PROGRAM o_Cons_Cmd_Actionneurs
VAR
	Calcul_Temp1: REAL;
	Mode_NEP_Chaud: BOOL;
	Mode_NEP_Froid: BOOL;
	Calcul_Debit_Bypass: REAL;
	ACH_Deb_Souf_Etat_Depol: REAL;
	ACH_Deb_Souf_Etat_Libre: REAL;
	ACH_Mode_Auto_Out_Debit_Souf: REAL;
	Consigne_Mode_EnFctnmnt_PD: REAL := 67.0;
	Consigne_Mode_EnFctnmnt_GD: REAL := 600.0;
END_VAR

(**********************************************Commande des actionneurs*)
Cmd_Appli_PC_Cab					:= (Mode_Auto.Cmd_Prise  AND Mode_Auto.Enable) OR (Mode_Manu.Cmd_Prise AND Mode_Manu.Enable);
Cmd_Appli_Vanne_Alim_Douche			:= (Mode_Auto.Cmd_Douche  AND Mode_Auto.Enable) OR (Mode_Manu.Cmd_Douche AND Mode_Manu.Enable) OR Forc_Ouv_Alim_Lav_Dou;
Cmd_Appli_Vanne_Alim_Douchette		:= ((Mode_Auto.Cmd_Douchette  AND Mode_Auto.Enable) OR (Mode_Manu.Cmd_Douchette AND Mode_Manu.Enable) OR Mode_Cabine_Nettoyage);
Cmd_Appli_Vanne_Alim_Lavabo			:= (Mode_Auto.Cmd_Lavabo  AND Mode_Auto.Enable) OR (Mode_Manu.Cmd_Lavabo AND Mode_Manu.Enable);
Cmd_Appli_Vanne_Vid_Douche			:= ((Mode_Auto.Cmd_Vidange_Douche  AND Mode_Auto.Enable) OR (Mode_Manu.Cmd_Vidange_Douche AND Mode_Manu.Enable) OR Mode_Cabine_Nettoyage);
Cmd_Appli_Vanne_Vid_Lavabo			:= ((Mode_Auto.Cmd_Vidange_Lavabo  AND Mode_Auto.Enable) OR (Mode_Manu.Cmd_Vidange_Lavabo AND Mode_Manu.Enable) OR Mode_Cabine_Nettoyage);
Cmd_Appli_ElectroValve_Alim_Douche	:= (Mode_Auto.Cmd_Electrovanne_Douche  AND Mode_Auto.Enable) OR (Mode_Manu.Cmd_Electrovanne_Douche AND Mode_Manu.Enable);
Cmd_Appli_ElectroValve_Alim_Lavabo	:= (Mode_Auto.Cmd_Electrovanne_Lavabo  AND Mode_Auto.Enable) OR (Mode_Manu.Cmd_Electrovanne_Lavabo AND Mode_Manu.Enable) OR Forc_Ouv_Alim_Lav_Dou;
Cmd_Appli_Reg_Etanche_Souf			:= (Cons_Actionneur_Registre_Souf_m3h > ((Cons_Max_Bas_Deb_Ext + 0.5) * Volume_Cabine)) AND Option_Reg_Etanche_Souf;
Cmd_Appli_Vanne_Alim_NEP			:=  (Mode_Auto.Cmd_NEP  AND Mode_Auto.Enable) OR (Mode_Manu.Cmd_NEP AND Mode_Manu.Enable);
Cmd_Appli_Verin_WC_GV				:=(Mode_Auto.Cmd_Verin_WC_GV  AND Mode_Auto.Enable) OR (Mode_Manu.Cmd_Verin_WC_GV AND Mode_Manu.Enable);
Cmd_Appli_Verin_WC_PV				:=(Mode_Auto.Cmd_Verin_WC_PV  AND Mode_Auto.Enable) OR (Mode_Manu.Cmd_Verin_WC_PV AND Mode_Manu.Enable);

(*Convertion des valeurs m3/h en Vol/h (ACH)*)
ACH_Deb_Souf_Etat_Depol 	:= Cons_Deb_Souf_Etat_Depol * Volume_Cabine;
ACH_Deb_Souf_Etat_Libre 	:= Cons_Deb_Souf_Etat_Libre * Volume_Cabine;
ACH_Mode_Auto_Out_Debit_Souf:= Mode_Auto.Out_Debit_Souf * Volume_Cabine;

(**********************************************Gestion de la consigne de débit en état cabine libre*)
IF(Mode_Cabine_Libre)
	THEN
	Cons_Actionneur_Registre_Ext_Volh 					:= ACH_Deb_Souf_Etat_Libre;
	Cons_Actionneur_Registre_Souf_Volh 					:= ACH_Deb_Souf_Etat_Libre;
	
	IF (ACH_Deb_Souf_Etat_Libre < 354.0) //Mettre la valeur maximum du débit du registre en diam 100mm
		THEN
		GVL_RegTROX.ConsAppliDeb_RegSouf_GD_FCVT01		:= 0.0;
		GVL_RegTROX.ConsAppliDeb_RegSouf_PD_FCVT02		:= ACH_Deb_Souf_Etat_Libre;
		ELSE
		GVL_RegTROX.ConsAppliDeb_RegSouf_GD_FCVT01		:= ACH_Deb_Souf_Etat_Libre;
		GVL_RegTROX.ConsAppliDeb_RegSouf_PD_FCVT02		:= 0.0;	
	END_IF
	GVL_RegTROX.ConsAppliDeb_RegSouf_Cabine_FCVT03		:= 1020.0; //Mettre le débit maximum pour qu'il reste ouvert à 100%
	GVL_RegTROX.ConsAppliDeb_Reg_Bypass_FCVT04			:= 0.0;
	GVL_RegTROX.ConsAppliDeb_RegSouf_CabGD_FCVT05		:= 0.0;
	GVL_RegTROX.ConsAppliDeb_RegSouf_CabPD_FCVT06		:= 0.0;
	GVL_RegTROX.ConsAppliDeb_RegRep_FCVT07				:= 0.0;
END_IF;

(**********************************************Gestion de la consigne de débit en etat cabine dépollution*)
IF(Mode_Cabine_Depollution OR Mode_Depollution_cycle1)
	THEN
	IF (Mode_Depollution_cycle1) // 1er cycle, décontamination de la CTA
		THEN
		Cons_Actionneur_Registre_Ext_Volh 					:= ACH_Deb_Souf_Etat_Depol;
		Cons_Actionneur_Registre_Souf_Volh 					:= ACH_Deb_Souf_Etat_Depol;
		
		GVL_RegTROX.ConsAppliDeb_RegSouf_GD_FCVT01			:= 375.0;
		GVL_RegTROX.ConsAppliDeb_RegSouf_PD_FCVT02			:= 100.0;
		GVL_RegTROX.ConsAppliDeb_RegSouf_Cabine_FCVT03		:= 0.0;
		GVL_RegTROX.ConsAppliDeb_Reg_Bypass_FCVT04			:= 0.0;
		GVL_RegTROX.ConsAppliDeb_RegSouf_CabGD_FCVT05		:= 575.0;
		GVL_RegTROX.ConsAppliDeb_RegSouf_CabPD_FCVT06		:= 100.0;
		GVL_RegTROX.ConsAppliDeb_RegRep_FCVT07				:= 200.0;
	END_IF;
	IF (Mode_Cabine_Depollution AND NOT Mode_Depollution_cycle1) // 2ème cycle, décontamination de la cabine
		THEN
		Cons_Actionneur_Registre_Ext_Volh 					:= ACH_Deb_Souf_Etat_Depol;
		Cons_Actionneur_Registre_Souf_Volh 					:= ACH_Deb_Souf_Etat_Depol;
		
		GVL_RegTROX.ConsAppliDeb_RegSouf_GD_FCVT01			:= ACH_Deb_Souf_Etat_Depol;
		GVL_RegTROX.ConsAppliDeb_RegSouf_PD_FCVT02			:= 0.0;
		GVL_RegTROX.ConsAppliDeb_RegSouf_Cabine_FCVT03		:= 1020.0; //Mettre le débit maximum pour qu'il reste ouvert à 100%
		GVL_RegTROX.ConsAppliDeb_Reg_Bypass_FCVT04			:= 0.0;
		GVL_RegTROX.ConsAppliDeb_RegSouf_CabGD_FCVT05		:= 0.0;
		GVL_RegTROX.ConsAppliDeb_RegSouf_CabPD_FCVT06		:= 0.0;
		GVL_RegTROX.ConsAppliDeb_RegRep_FCVT07				:= 0.0;
	END_IF;
END_IF;

(**********************************************Gestion de la consigne de débit en etat cabine Mode mise en condition*)
IF(Mode_MEnCond AND NOT Mode_Cabine_Libre)
	THEN
	Cons_Actionneur_Registre_Ext_Volh 					:= ACH_Mode_Auto_Out_Debit_Souf;
	Cons_Actionneur_Registre_Souf_Volh 					:= ACH_Mode_Auto_Out_Debit_Souf;
	
	GVL_RegTROX.ConsAppliDeb_RegSouf_GD_FCVT01			:= 0.0;
	GVL_RegTROX.ConsAppliDeb_RegSouf_PD_FCVT02			:= 0.0;
	GVL_RegTROX.ConsAppliDeb_RegSouf_Cabine_FCVT03		:= 0.0;
	GVL_RegTROX.ConsAppliDeb_Reg_Bypass_FCVT04			:= 0.0;
	IF (ACH_Mode_Auto_Out_Debit_Souf < 354.0)  //Mettre la valeur maximum du débit du registre en diam 100mm
		THEN
		GVL_RegTROX.ConsAppliDeb_RegSouf_CabGD_FCVT05	:= 0.0;
		GVL_RegTROX.ConsAppliDeb_RegSouf_CabPD_FCVT06	:= ACH_Mode_Auto_Out_Debit_Souf;
		ELSE
		GVL_RegTROX.ConsAppliDeb_RegSouf_CabGD_FCVT05	:= ACH_Mode_Auto_Out_Debit_Souf;
		GVL_RegTROX.ConsAppliDeb_RegSouf_CabPD_FCVT06	:= 0.0;	
	END_IF
	GVL_RegTROX.ConsAppliDeb_RegRep_FCVT07				:= 1020.0; //Mettre le débit maximum pour qu'il reste ouvert à 100%
END_IF;

(**********************************************Gestion de la consigne de débit en etat cabine Mode fonctionnement*)
IF(Mode_Fctnmt AND NOT Mode_Cabine_Libre)
	THEN
	Cons_Actionneur_Registre_Ext_Volh 					:= ACH_Mode_Auto_Out_Debit_Souf;
	Cons_Actionneur_Registre_Souf_Volh 					:= ACH_Mode_Auto_Out_Debit_Souf;
	(*IF (ACH_Mode_Auto_Out_Debit_Souf < 354.0) //Mettre la valeur maximum du débit du registre en diam 100mm
		THEN
		GVL_RegTROX.ConsAppliDeb_RegSouf_GD_FCVT01		:= 0.0;
		GVL_RegTROX.ConsAppliDeb_RegSouf_PD_FCVT02		:= ACH_Mode_Auto_Out_Debit_Souf;
		ELSE
		GVL_RegTROX.ConsAppliDeb_RegSouf_GD_FCVT01		:= ACH_Mode_Auto_Out_Debit_Souf;
		GVL_RegTROX.ConsAppliDeb_RegSouf_PD_FCVT02		:= 0.0;	
	END_IF*)
	GVL_RegTROX.ConsAppliDeb_RegSouf_GD_FCVT01			:= 0.0;
	GVL_RegTROX.ConsAppliDeb_RegSouf_PD_FCVT02			:= ACH_Mode_Auto_Out_Debit_Souf;
	GVL_RegTROX.ConsAppliDeb_RegSouf_Cabine_FCVT03		:= 0.0;
	Calcul_Debit_Bypass 								:= LIMIT(0.0, 600.0 - (Consigne_Mode_EnFctnmnt_GD + ACH_Mode_Auto_Out_Debit_Souf), 579.0);
	GVL_RegTROX.ConsAppliDeb_Reg_Bypass_FCVT04			:= Calcul_Debit_Bypass;
	GVL_RegTROX.ConsAppliDeb_RegSouf_CabGD_FCVT05		:= Consigne_Mode_EnFctnmnt_GD;
	GVL_RegTROX.ConsAppliDeb_RegSouf_CabPD_FCVT06		:= 0.0;
	(*IF (ACH_Mode_Auto_Out_Debit_Souf < 354.0) //Mettre la valeur maximum du débit du registre en diam 100mm
		THEN
		GVL_RegTROX.ConsAppliDeb_RegSouf_CabGD_FCVT05	:= 0.0;
		GVL_RegTROX.ConsAppliDeb_RegSouf_CabPD_FCVT06	:= ACH_Mode_Auto_Out_Debit_Souf;
		ELSE
		GVL_RegTROX.ConsAppliDeb_RegSouf_CabGD_FCVT05	:= ACH_Mode_Auto_Out_Debit_Souf;
		GVL_RegTROX.ConsAppliDeb_RegSouf_CabPD_FCVT06	:= 0.0;	
	END_IF*)
	GVL_RegTROX.ConsAppliDeb_RegRep_FCVT07				:= LIMIT(0, Consigne_Mode_EnFctnmnt_GD - ACH_Mode_Auto_Out_Debit_Souf, 1020.0);
END_IF;

(**********************************************Consigne des actionneurs en mode manuel*)
IF(Mode_Cabine_Manuel)
	THEN
	Cons_Actionneur_Registre_Ext_Volh 					:= Cons_Deb_Soufflage_Appli;
	Cons_Actionneur_Registre_Souf_Volh 					:= Cons_Deb_Soufflage_Appli;
	IF (Cons_Deb_Soufflage_Appli < 354.0) //Mettre la valeur maximum du débit du registre en diam 100mm
		THEN
		GVL_RegTROX.ConsAppliDeb_RegSouf_GD_FCVT01		:= 0.0;
		GVL_RegTROX.ConsAppliDeb_RegSouf_PD_FCVT02		:= Cons_Deb_Soufflage_Appli;
		ELSE
		GVL_RegTROX.ConsAppliDeb_RegSouf_GD_FCVT01		:= Cons_Deb_Soufflage_Appli;
		GVL_RegTROX.ConsAppliDeb_RegSouf_PD_FCVT02		:= 0.0;	
	END_IF
	GVL_RegTROX.ConsAppliDeb_RegSouf_Cabine_FCVT03		:= 0.0;
	GVL_RegTROX.ConsAppliDeb_Reg_Bypass_FCVT04			:= 0.0;
	GVL_RegTROX.ConsAppliDeb_RegSouf_CabGD_FCVT05		:= 0.0;
	GVL_RegTROX.ConsAppliDeb_RegSouf_CabPD_FCVT06		:= 0.0;
	GVL_RegTROX.ConsAppliDeb_RegRep_FCVT07				:= 0.0;
END_IF;

(**********************************************Gestion des consignes en cas de défaut sur le capteur de pression*)
IF (Defaut_Sonde_Press_Cabine AND NOT Dmd_Post_Ventilation)
	THEN
	GVL_RegTROX.ConsAppliDeb_RegSouf_GD_FCVT01			:= 0.0;
	GVL_RegTROX.ConsAppliDeb_RegSouf_PD_FCVT02			:= 0.0;	
	GVL_RegTROX.ConsAppliDeb_RegSouf_Cabine_FCVT03		:= 0.0;
	GVL_RegTROX.ConsAppliDeb_Reg_Bypass_FCVT04			:= 0.0;
	GVL_RegTROX.ConsAppliDeb_RegSouf_CabGD_FCVT05		:= 0.0;
	GVL_RegTROX.ConsAppliDeb_RegSouf_CabPD_FCVT06		:= 0.0;
	GVL_RegTROX.ConsAppliDeb_RegRep_FCVT07				:= 0.0;
END_IF

(**********************************************Consigne des actionneurs en mode automatique*)
IF(Mode_Cabine_Automatique AND NOT Mode_Cabine_Depollution AND NOT Mode_MEnCond AND NOT Mode_Fctnmt)
	THEN
	Cons_Actionneur_Registre_Ext_Volh	:= Cons_Deb_Soufflage_Appli;
	Cons_Actionneur_Registre_Souf_Volh	:= Cons_Deb_Soufflage_Appli;
	Cons_Actionneur_Moteur_ByPass		:= Mode_Auto.Out_Cons_Moteur_ByPass;
	// Deux types de fonctionnement, la première si une reccette est déclaré avec une gestion de CTA et le deuxième type sans gestion de CTA
	IF (RS_MEnCond.Q1)// gestion avec CTA (Activation des redistres de soufflage générale et du soufflage de la cabine)
		THEN
		Cons_Actionneur_Registre_Ext_Volh 					:= ACH_Mode_Auto_Out_Debit_Souf;
		Cons_Actionneur_Registre_Souf_Volh 					:= ACH_Mode_Auto_Out_Debit_Souf;
		(*IF (ACH_Mode_Auto_Out_Debit_Souf < 354.0) //Mettre la valeur maximum du débit du registre en diam 100mm
			THEN
			GVL_RegTROX.ConsAppliDeb_RegSouf_GD_FCVT01		:= 0.0;
			GVL_RegTROX.ConsAppliDeb_RegSouf_PD_FCVT02		:= ACH_Mode_Auto_Out_Debit_Souf;
			ELSE
			GVL_RegTROX.ConsAppliDeb_RegSouf_GD_FCVT01		:= ACH_Mode_Auto_Out_Debit_Souf;
			GVL_RegTROX.ConsAppliDeb_RegSouf_PD_FCVT02		:= 0.0;	
		END_IF*)
		GVL_RegTROX.ConsAppliDeb_RegSouf_GD_FCVT01			:= 0.0;
		GVL_RegTROX.ConsAppliDeb_RegSouf_PD_FCVT02			:= Consigne_Mode_EnFctnmnt_PD;
		GVL_RegTROX.ConsAppliDeb_RegSouf_Cabine_FCVT03		:= 0.0;
		Calcul_Debit_Bypass 								:= LIMIT(0.0, 600.0 - (Consigne_Mode_EnFctnmnt_GD + Consigne_Mode_EnFctnmnt_PD), 579.0);
		GVL_RegTROX.ConsAppliDeb_Reg_Bypass_FCVT04			:= Calcul_Debit_Bypass;
		GVL_RegTROX.ConsAppliDeb_RegSouf_CabGD_FCVT05		:= Consigne_Mode_EnFctnmnt_GD;
		GVL_RegTROX.ConsAppliDeb_RegSouf_CabPD_FCVT06		:= 0.0;
		(*IF (ACH_Mode_Auto_Out_Debit_Souf < 354.0) //Mettre la valeur maximum du débit du registre en diam 100mm
			THEN
			GVL_RegTROX.ConsAppliDeb_RegSouf_CabGD_FCVT05	:= 0.0;
			GVL_RegTROX.ConsAppliDeb_RegSouf_CabPD_FCVT06	:= ACH_Mode_Auto_Out_Debit_Souf;
			ELSE
			GVL_RegTROX.ConsAppliDeb_RegSouf_CabGD_FCVT05	:= ACH_Mode_Auto_Out_Debit_Souf;
			GVL_RegTROX.ConsAppliDeb_RegSouf_CabPD_FCVT06	:= 0.0;	
		END_IF*)
		GVL_RegTROX.ConsAppliDeb_RegRep_FCVT07				:= LIMIT(0, Consigne_Mode_EnFctnmnt_GD - Consigne_Mode_EnFctnmnt_PD, 1020.0);
	ELSE // gestion sans CTA (Activation des redistres de soufflage générale uniquement et ouverture du registre FCVT03)
		IF (Cons_Deb_Soufflage_Appli < 354.0) //Mettre la valeur maximum du débit du registre en diam 100mm
			THEN
			GVL_RegTROX.ConsAppliDeb_RegSouf_GD_FCVT01		:= 0.0;
			GVL_RegTROX.ConsAppliDeb_RegSouf_PD_FCVT02		:= Cons_Deb_Soufflage_Appli;
			ELSE
			GVL_RegTROX.ConsAppliDeb_RegSouf_GD_FCVT01		:= Cons_Deb_Soufflage_Appli;
			GVL_RegTROX.ConsAppliDeb_RegSouf_PD_FCVT02		:= 0.0;	
		END_IF
		GVL_RegTROX.ConsAppliDeb_RegSouf_Cabine_FCVT03		:= 1020.0; //Mettre le débit maximum pour qu'il reste ouvert à 100%
		GVL_RegTROX.ConsAppliDeb_Reg_Bypass_FCVT04			:= 0.0;
		GVL_RegTROX.ConsAppliDeb_RegSouf_CabGD_FCVT05		:= 0.0;
		GVL_RegTROX.ConsAppliDeb_RegSouf_CabPD_FCVT06		:= 0.0;
		GVL_RegTROX.ConsAppliDeb_RegRep_FCVT07				:= 0.0;
	END_IF
END_IF;

(**********************************************Gestion de la consigne de température, de débit soufflage et de débit extraction en etat cabine nettoyage vol/h*)
IF(Mode_Cabine_Nettoyage)
	THEN
	Cons_Actionneur_Registre_Ext_Volh := Cons_Deb_Souf_Etat_Nettoyage;
	Cons_Actionneur_Registre_Souf_Volh := Cons_Deb_Souf_Etat_Nettoyage;
END_IF;

(**********************************************Gestion de la consigne de température, de débit soufflage et de débit extraction en etat cabine evaluation vol/h*)
IF(Mode_Evaluation)
	THEN
	Cons_Actionneur_Registre_Ext_Volh := Cons_Deb_Souf_Etat_Evaluation;
	Cons_Actionneur_Registre_Souf_Volh := Cons_Deb_Souf_Etat_Evaluation;
END_IF;

(**********************************************Consigne de la vanne 3 voies eau mitigée*)
(*Deux types de gestion, une via la regul PID si une vanne d'alimentation est ouverte et la deuxième si il y'a la NEP (Position de régulation au repos)*)
Mode_NEP_Chaud := Mode_Auto.Mode_18 OR Mode_Manu.Mode_18;
Mode_NEP_Froid := Mode_Auto.Mode_19 OR Mode_Manu.Mode_19;

IF(Mode_NEP_Chaud OR Mode_NEP_Froid)
	THEN
	Cons_Actionneur_V3V_Eau_Mitig := MAX(Mode_Auto.Out_Cons_V3V_Eau_Mitig , Mode_Manu.Out_Cons_V3V_Eau_Mitig);
	ELSE
	Cons_Actionneur_V3V_Eau_Mitig := S_Cmd_PID_Temp_Eau_Mitig;
END_IF;

(**********************************************Forçage ouverture electrovanne lavabo et douche pour eviter l'achéssement*******************************************************************************)
IF((Mode_Cabine_Libre AND Option_Cabine_Humide AND ((VDayOfWeek = Cons_J_Forc_Vid_Lavabo) AND (Vheure = Cons_H_Forc_Vid_Lavabo) AND (Vminute = Cons_M_Forc_Vid_Lavabo))))
	THEN
	Forc_Ouv_Alim_Lav_Dou := FALSE;
	ELSE
	Forc_Ouv_Alim_Lav_Dou := FALSE;
END_IF;

(**********************************************Convertion en m3/h pour la consigne de soufflage et d'extraction******************************************)
Cons_Actionneur_Registre_Ext_m3h := (Cons_Actionneur_Registre_Ext_Volh * Volume_Cabine);
Cons_Actionneur_Registre_Souf_m3h := (Cons_Actionneur_Registre_Souf_Volh * Volume_Cabine);

(**********************************************Convertion en °F pour la consigne de la vanne thermo******************************************)
Calcul_Temp1 := ((1.8 * Cons_Temperature_Eau) + 32.0);
Cons_Temperature_Eau_F := REAL_TO_INT(Calcul_Temp1 * 10);

(**********************************************Consigne appliquée sur le registre étanche d'extraction******************************************)
IF (Option_Reg_Etanche_Ext)
	THEN
	IF(Option_Regul_Deb_Ou_Press)
		THEN
		Cons_Actionneur_Reg_Etanche_Ext := S_Cmd_PID_Press_Cab;
		ELSE
		IF((Cons_Actionneur_Registre_Ext_m3h > ((Cons_Max_Bas_Deb_Ext + 0.5) * Volume_Cabine)))
			THEN
			Cons_Actionneur_Reg_Etanche_Ext := 100.0;
			ELSE
			Cons_Actionneur_Reg_Etanche_Ext := 0.0;
		END_IF;
	END_IF;
ELSE
	Cons_Actionneur_Reg_Etanche_Ext := 0.0;
END_IF;

(**********************************************Gestion de la consigne de débit en mode post ventilation*)
IF(Dmd_Post_Ventilation)
	THEN
	Cons_Actionneur_Registre_Ext_Volh 					:= 0.0;
	Cons_Actionneur_Registre_Souf_Volh 					:= 0.0;
	
	GVL_RegTROX.ConsAppliDeb_RegSouf_GD_FCVT01			:= 675.0;
	GVL_RegTROX.ConsAppliDeb_RegSouf_PD_FCVT02			:= 0.0;
	GVL_RegTROX.ConsAppliDeb_RegSouf_Cabine_FCVT03		:= 0.0;
	GVL_RegTROX.ConsAppliDeb_Reg_Bypass_FCVT04			:= 0.0;
	GVL_RegTROX.ConsAppliDeb_RegSouf_CabGD_FCVT05		:= 675.0;
	GVL_RegTROX.ConsAppliDeb_RegSouf_CabPD_FCVT06		:= 0.0;
	GVL_RegTROX.ConsAppliDeb_RegRep_FCVT07				:= 0.0;
END_IF;

(**********************************************Déclaration des VAV en communication******************************************)
(**********************************************VAV FCVT01*)
(*Sonde*)
GVL_RegTROX.MES_RegSouf_GD_FCVT01(
	Enable_Alarme:= TRUE, 
	Status_DEF_EAN:= GVL_RegTROX.RegSouf_GD_FCVT01_DefCom OR GVL_RegTROX.RegSouf_GD_FCVT01_Def_DiscordDeb, 
	Tempo_AL:= T#10S, 
	EAN_MIN:= 0.0, 
	EAN_MAX:= 1020.0, 
	MES_MIN:= 0.0, 
	MES_MAX:= 1020.0, 
	Filtre_Actif:= FALSE, 
	Temps_Echantillonage:= T#500MS, 
	Tab_Sonde:= GVL_RegTROX.TAB_Sonde_RegSouf_GD_FCVT01);
(*Registre*)	
GVL_RegTROX.RegSouf_GD_FCVT01(
	Cons_Pos_Dem:= GVL_RegTROX.Com_RegSouf_GD_FCVT01.MES_Pos, 
	Type_Consigne:= TRUE, 
	Control_Discordance:= FALSE, 
	Presence_Fdc:= 0, 
	Inverse_SAN:= FALSE, 
	SAN_MIN:= 0.0, 
	SAN_MAX:= 1020.0,
	Tab_RegMoto:= GVL_RegTROX.TAB_Reg_RegSouf_GD_FCVT01);
	
(**********************************************VAV FCVT02*)
(*Sonde*)
GVL_RegTROX.MES_RegSouf_PD_FCVT02(
	Enable_Alarme:= TRUE, 
	Status_DEF_EAN:= GVL_RegTROX.RegSouf_PD_FCVT02_DefCom OR GVL_RegTROX.RegSouf_PD_FCVT02_Def_DiscordDeb, 
	Tempo_AL:= T#10S, 
	EAN_MIN:= 0.0, 
	EAN_MAX:= 364.0, 
	MES_MIN:= 0.0, 
	MES_MAX:= 364.0, 
	Filtre_Actif:= FALSE, 
	Temps_Echantillonage:= T#500MS, 
	Tab_Sonde:= GVL_RegTROX.TAB_Sonde_RegSouf_PD_FCVT02);
(*Registre*)	
GVL_RegTROX.RegSouf_PD_FCVT02(
	Cons_Pos_Dem:= GVL_RegTROX.Com_RegSouf_PD_FCVT02.MES_Pos, 
	Type_Consigne:= TRUE, 
	Control_Discordance:= FALSE, 
	Presence_Fdc:= 0, 
	Inverse_SAN:= FALSE, 
	SAN_MIN:= 0.0, 
	SAN_MAX:= 364.0,
	Tab_RegMoto:= GVL_RegTROX.TAB_Reg_RegSouf_PD_FCVT02);

(**********************************************VAV FCVT03*)
(*Sonde*)
GVL_RegTROX.MES_RegSouf_Cabine_FCVT03(
	Enable_Alarme:= TRUE, 
	Status_DEF_EAN:= GVL_RegTROX.RegSouf_Cabine_FCVT03_DefCom, 
	Tempo_AL:= T#10S, 
	EAN_MIN:= 0.0, 
	EAN_MAX:= 1020.0, 
	MES_MIN:= 0.0, 
	MES_MAX:= 1020.0, 
	Filtre_Actif:= FALSE, 
	Temps_Echantillonage:= T#500MS, 
	Tab_Sonde:= GVL_RegTROX.TAB_Sonde_RegSouf_Cabine_FCVT03);
(*Registre*)	
GVL_RegTROX.RegSouf_Cabine_FCVT03(
	Cons_Pos_Dem:= GVL_RegTROX.Com_RegSouf_Cabine_FCVT03.MES_Pos, 
	Type_Consigne:= TRUE, 
	Control_Discordance:= FALSE, 
	Presence_Fdc:= 0, 
	Inverse_SAN:= FALSE, 
	SAN_MIN:= 0.0, 
	SAN_MAX:= 1020.0,
	Tab_RegMoto:= GVL_RegTROX.TAB_Reg_RegSouf_Cabine_FCVT03);

(**********************************************VAV FCVT04*)
(*Sonde*)
GVL_RegTROX.MES_RegBypass_FCVT04(
	Enable_Alarme:= TRUE, 
	Status_DEF_EAN:= GVL_RegTROX.Reg_Bypass_FCVT04_DefCom OR GVL_RegTROX.Reg_Bypass_FCVT04_Def_DiscordDeb, 
	Tempo_AL:= T#10S, 
	EAN_MIN:= 0.0, 
	EAN_MAX:= 579.0, 
	MES_MIN:= 0.0, 
	MES_MAX:= 579.0, 
	Filtre_Actif:= FALSE, 
	Temps_Echantillonage:= T#500MS, 
	Tab_Sonde:= GVL_RegTROX.TAB_Sonde_RegBypass_FCVT04);
(*Registre*)	
GVL_RegTROX.RegBypass_FCVT04(
	Cons_Pos_Dem:= GVL_RegTROX.Com_Reg_Bypass_FCVT04.MES_Pos, 
	Type_Consigne:= TRUE, 
	Control_Discordance:= FALSE, 
	Presence_Fdc:= 0, 
	Inverse_SAN:= FALSE, 
	SAN_MIN:= 0.0, 
	SAN_MAX:= 579.0,
	Tab_RegMoto:= GVL_RegTROX.TAB_Reg_RegBypass_FCVT04);
	
(**********************************************VAV FCVT05*)
(*Sonde*)
GVL_RegTROX.MES_RegSouf_CabGD_FCVT05(
	Enable_Alarme:= TRUE, 
	Status_DEF_EAN:= GVL_RegTROX.RegSouf_CabGD_FCVT05_DefCom OR GVL_RegTROX.RegSouf_CabGD_FCVT05_Def_DiscordDeb, 
	Tempo_AL:= T#10S, 
	EAN_MIN:= 0.0, 
	EAN_MAX:= 1020.0, 
	MES_MIN:= 0.0, 
	MES_MAX:= 1020.0, 
	Filtre_Actif:= FALSE, 
	Temps_Echantillonage:= T#500MS, 
	Tab_Sonde:= GVL_RegTROX.TAB_Sonde_RegSouf_CabGD_FCVT05);
(*Registre*)	
GVL_RegTROX.RegSouf_CabGD_FCVT05(
	Cons_Pos_Dem:= GVL_RegTROX.Com_RegSouf_CabGD_FCVT05.MES_Pos, 
	Type_Consigne:= TRUE, 
	Control_Discordance:= FALSE, 
	Presence_Fdc:= 0, 
	Inverse_SAN:= FALSE, 
	SAN_MIN:= 0.0, 
	SAN_MAX:= 1020.0,
	Tab_RegMoto:= GVL_RegTROX.TAB_Reg_RegSouf_CabGD_FCVT05);
	
(**********************************************VAV FCVT06*)
(*Sonde*)
GVL_RegTROX.MES_RegSouf_CabPD_FCVT06(
	Enable_Alarme:= TRUE, 
	Status_DEF_EAN:= GVL_RegTROX.RegSouf_CabPD_FCVT06_DefCom OR GVL_RegTROX.RegSouf_CabPD_FCVT06_Def_DiscordDeb, 
	Tempo_AL:= T#10S, 
	EAN_MIN:= 0.0, 
	EAN_MAX:= 364.0, 
	MES_MIN:= 0.0, 
	MES_MAX:= 364.0, 
	Filtre_Actif:= FALSE, 
	Temps_Echantillonage:= T#500MS, 
	Tab_Sonde:= GVL_RegTROX.TAB_Sonde_RegSouf_CabPD_FCVT06);
(*Registre*)	
GVL_RegTROX.RegSouf_CabPD_FCVT06(
	Cons_Pos_Dem:= GVL_RegTROX.Com_RegSouf_CabPD_FCVT06.MES_Pos, 
	Type_Consigne:= TRUE, 
	Control_Discordance:= FALSE, 
	Presence_Fdc:= 0, 
	Inverse_SAN:= FALSE, 
	SAN_MIN:= 0.0, 
	SAN_MAX:= 364.0,
	Tab_RegMoto:= GVL_RegTROX.TAB_Reg_RegSouf_CabPD_FCVT06);
	
(**********************************************VAV FCVT07*)
(*Sonde*)
GVL_RegTROX.MES_RegRep_FCVT07(
	Enable_Alarme:= TRUE, 
	Status_DEF_EAN:= GVL_RegTROX.RegRep_FCVT07_DefCom, 
	Tempo_AL:= T#10S, 
	EAN_MIN:= 0.0, 
	EAN_MAX:= 1020.0, 
	MES_MIN:= 0.0, 
	MES_MAX:= 1020.0, 
	Filtre_Actif:= FALSE, 
	Temps_Echantillonage:= T#500MS, 
	Tab_Sonde:= GVL_RegTROX.TAB_Sonde_RegRep_FCVT07);
(*Registre*)	
GVL_RegTROX.RegRep_FCVT07(
	Cons_Pos_Dem:= GVL_RegTROX.Com_RegRep_FCVT07.MES_Pos, 
	Type_Consigne:= TRUE, 
	Control_Discordance:= FALSE, 
	Presence_Fdc:= 0, 
	Inverse_SAN:= FALSE, 
	SAN_MIN:= 0.0, 
	SAN_MAX:= 1020.0,
	Tab_RegMoto:= GVL_RegTROX.TAB_Reg_RegRep_FCVT07);

END_PROGRAM

(* stored: Version 1.1.0.1, ProductVersion 3.1.4024.16
   POU o_Cons_Cmd_Actionneurs: Id {6c54e938-1130-4058-9ae4-db92486b75e2}, SpecialFunc None *)
